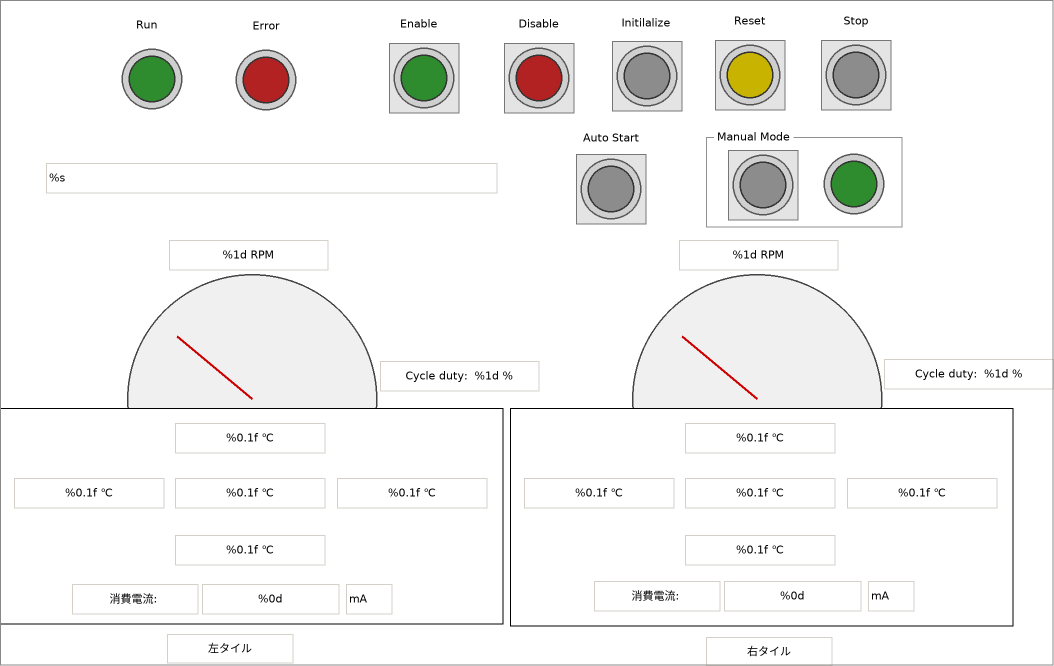
VISUALIZATION Visualization_operation  // 1054x666
    Group (0,0 1054x666)
        PushSwitch (389,43 70x70), variable: MAIN.bEnable, behaviour: TAP, style: Switch-PushSwitch-Green
        Label (369,9 100x30), "Enable"
        PushSwitch (504,43 70x70), variable: MAIN.bDisable, behaviour: TAP, style: Switch-PushSwitch-Red
        Label (489,9 100x30), "Disable"
        Lamp1 (117,44 70x70), variable: MAIN.ServoON, style: Lamp-Lamp1-Green
        Lamp1 (231,45 70x70), variable: MAIN.Error, style: Lamp-Lamp1-Red
        Label (97,0 100x50), "Run"
        Label (216,1 100x50), "Error"
        PushSwitch (715,40 70x70), variable: MAIN.bReset, behaviour: TAP, style: Switch-PushSwitch-Yellow
        Label (700,6 100x30), "Reset"
        PushSwitch (821,40 70x70), variable: MAIN.bStop, behaviour: TAP, style: Switch-PushSwitch-Gray
        Label (806,6 100x30), "Stop"
        Meter180 (632,274 250x250), value: IoT.planar_tiles_diag_data[1].fan_rpm, style: Meter-Meter180-Gray, scale format: %1d, scale 0..3000
        Meter180 (127,274 250x250), value: IoT.planar_tiles_diag_data[2].fan_rpm, style: Meter-Meter180-Gray, scale format: %1d, scale 0..3000
        RoundedRectangle (0,408 503x216)
        Textfield (14,478 150x30), "%0.1f ℃", text variable: IoT.planar_tiles_diag_data[2].temperature_west / 10
        Textfield (175,478 150x30), "%0.1f ℃", text variable: IoT.planar_tiles_diag_data[2].temperature_center / 10
        Textfield (337,478 150x30), "%0.1f ℃", text variable: IoT.planar_tiles_diag_data[2].temperature_east / 10
        Textfield (175,423 150x30), "%0.1f ℃", text variable: IoT.planar_tiles_diag_data[2].temperature_north / 10
        Textfield (175,535 150x30), "%0.1f ℃", text variable: IoT.planar_tiles_diag_data[2].temperature_south / 10
        RoundedRectangle (510,408 503x218)
        Textfield (524,478 150x30), "%0.1f ℃", text variable: IoT.planar_tiles_diag_data[1].temperature_west / 10
        Textfield (685,478 150x30), "%0.1f ℃", text variable: IoT.planar_tiles_diag_data[1].temperature_center / 10
        Textfield (847,478 150x30), "%0.1f ℃", text variable: IoT.planar_tiles_diag_data[1].temperature_east / 10
        Textfield (685,423 150x30), "%0.1f ℃", text variable: IoT.planar_tiles_diag_data[1].temperature_north / 10
        Textfield (685,535 150x30), "%0.1f ℃", text variable: IoT.planar_tiles_diag_data[1].temperature_south / 10
        Textfield (202,584 137x30), "%0d", text variable: IoT.planar_tiles_diag_data[2].power_supply_current / 10
        Textfield (72,584 126x30), "消費電流:"
        Textfield (346,584 46x30), "mA"
        Textfield (724,581 137x30), "%0d", text variable: IoT.planar_tiles_diag_data[1].power_supply_current / 10
        Textfield (594,581 126x30), "消費電流:"
        Textfield (868,581 46x30), "mA"
        Textfield (706,637 126x29), "右タイル"
        Textfield (167,634 126x29), "左タイル"
        Textfield (380,361 159x30), "Cycle duty: %1d %", text variable: IoT.planar_tiles_diag_data[2].fan_duty_cycle
        Textfield (884,359 170x30), "Cycle duty: %1d %", text variable: IoT.planar_tiles_diag_data[2].fan_duty_cycle
        Textfield (169,240 159x30), "%1d RPM", text variable: IoT.planar_tiles_diag_data[2].fan_rpm
        Textfield (679,240 159x30), "%1d RPM", text variable: IoT.planar_tiles_diag_data[1].fan_rpm
        Textfield (46,163 451x30), "%s", text variable: MAIN.ads_reporter.executing.task_name
        PushSwitch (612,41 70x70), variable: MAIN.Init_Start, behaviour: TOGGLE, style: Switch-PushSwitch-Gray
        Label (596,8 100x30), "Initilalize"
        PushSwitch (576,154 70x70), variable: MAIN.Demo_Start, behaviour: TOGGLE, style: Switch-PushSwitch-Gray
        Label (561,123 100x30), "Auto Start"
        GroupBox (706,129 196x98), "Manual Mode"
            Lamp1 (113,20 70x70), variable: MAIN.manu_mode, style: Lamp-Lamp1-Green
            PushSwitch (22,21 70x70), variable: MAIN.manu_mode, behaviour: TOGGLE, style: Switch-PushSwitch-Gray
        Lamp1 (819,149 70x70), variable: MAIN.manu_mode, style: Lamp-Lamp1-Green
        PushSwitch (728,150 70x70), variable: MAIN.manu_mode, behaviour: TOGGLE, style: Switch-PushSwitch-Gray
END_VISUALIZATION

(* stored: Version 1.1.0.1, ProductVersion 3.1.4024.12
   Visu Visualization_operation: Id {799ca28c-2efc-4fc9-97c1-20fb5bd34753} *)
